{attribute 'GeneratedUsingTerminal: EL3423-0000-0020'}
{attribute addProperty BoxType "EL3423-0000-0020"}
{attribute addProperty Id "Active_EnergyAT %I*LINT8"}
{attribute addProperty CRC "241265381"}
{attribute addProperty Size "8"}
TYPE Total_Active_Reduced_0E616AE5 :
STRUCT
	{attribute addProperty Name "Active_Energy"}
	Active_Energy AT %I* : LINT;
END_STRUCT
END_TYPE

(* stored: Version 1.2.0.0, ProductVersion 3.1.4024.9
   DUT Total_Active_Reduced_0E616AE5: Id {db296974-cede-426e-ab9b-6cb35ab632e3} *)
